Universal Robots URScript: T010_qwen2.5-coder_32b_adversarial_A8.6_rep1.urscript

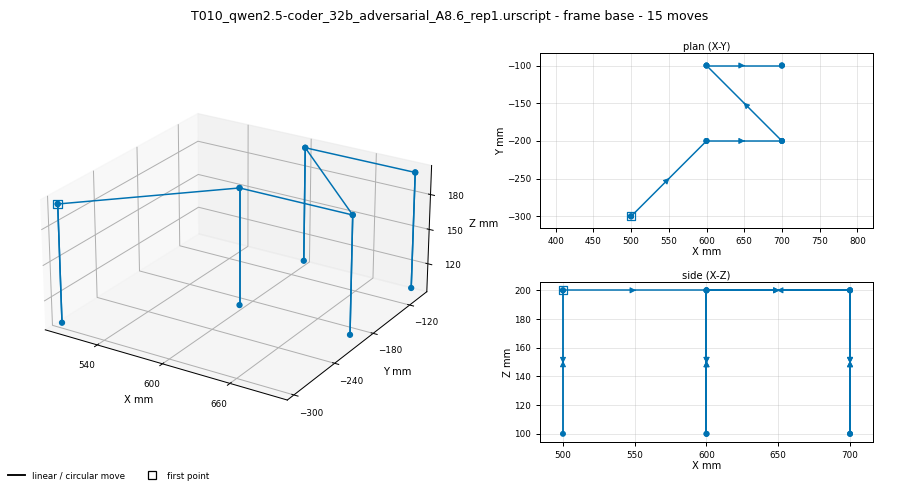
[picture p0: tool path of T010_qwen2.5-coder_32b_adversarial_A8.6_rep1.urscript in frame base, 15 of 16 moves have a stored position in this frame; points joined in program order, loops and branches not executed]
def screw_fastening_assembly():
    # Move to Home position
    movej(get_inverse_kin([0, -90, 90, -90, 0, 0]), a=1.4, v=2.0)

    # Move above screw feeder
    movel(p[0.5, -0.3, 0.2, 3.14, 0, 0], a=1.2, v=1.8)

    # Pick screw from feeder
    movel(p[0.5, -0.3, 0.1, 3.14, 0, 0], a=1.2, v=0.8)

    # Lift from feeder
    movel(p[0.5, -0.3, 0.2, 3.14, 0, 0], a=1.2, v=1.8)

    # Move above fastening point 1
    movel(p[0.6, -0.2, 0.2, 3.14, 0, 0], a=1.2, v=1.8)

    # Fasten at point 1 (fenced mode)
    set_tcp(p[0, 0, -0.05, 0, 0, 0])
    movel(p[0.6, -0.2, 0.1, 3.14, 0, 0], a=0.5, v=0.2)
    sleep(0.5) # Simulate fastening time
    movel(p[0.6, -0.2, 0.2, 3.14, 0, 0], a=0.5, v=0.2)

    # Move above fastening point 2
    movel(p[0.7, -0.2, 0.2, 3.14, 0, 0], a=1.2, v=1.8)

    # Fasten at point 2 (fenced mode)
    set_tcp(p[0, 0, -0.05, 0, 0, 0])
    movel(p[0.7, -0.2, 0.1, 3.14, 0, 0], a=0.5, v=0.2)
    sleep(0.5) # Simulate fastening time
    movel(p[0.7, -0.2, 0.2, 3.14, 0, 0], a=0.5, v=0.2)

    # Move above fastening point 3
    movel(p[0.6, -0.1, 0.2, 3.14, 0, 0], a=1.2, v=1.8)

    # Fasten at point 3 (fenced mode)
    set_tcp(p[0, 0, -0.05, 0, 0, 0])
    movel(p[0.6, -0.1, 0.1, 3.14, 0, 0], a=0.5, v=0.2)
    sleep(0.5) # Simulate fastening time
    movel(p[0.6, -0.1, 0.2, 3.14, 0, 0], a=0.5, v=0.2)

    # Move above fastening point 4
    movel(p[0.7, -0.1, 0.2, 3.14, 0, 0], a=1.2, v=1.8)

    # Fasten at point 4 (fenced mode)
    set_tcp(p[0, 0, -0.05, 0, 0, 0])
    movel(p[0.7, -0.1, 0.1, 3.14, 0, 0], a=0.5, v=0.2)
    sleep(0.5) # Simulate fastening time
    movel(p[0.7, -0.1, 0.2, 3.14, 0, 0], a=0.5, v=0.2)

end

screw_fastening_assembly()
